(* Logix 5000 project; controller Reto2 vendor 1 type 14 code 156 rev 30.11; software revision 30.00 *)

TASK MainTask (continuous, watchdog 500 ms) : MainProgram

MODULES
   Local : vendor 1 type 14 code 156 (Compact 0, rev 30.11)
      Digital_IN : 1769-IQ16 (Compact 4, rev 1.1, Input RPI 20 ms)
      Digital_OUT : vendor 1 type 7 code 86 (Compact 5, rev 2.1, Output RPI 20 ms)
END_MODULES

VAR_GLOBAL   (* controller tags *)
   AUTO : BOOL;   // Switch Auto FactoryIO
   BOX_AT_ENTRY : BOOL := 1;   // Sensor cajas FactoryIO
   BOX_FEEDER : BOOL;   // Banda 1 cajas FactoryIO
   CLAMP : BOOL;   // Palanca junta cajas FactoryIO
   CLAMPED : BOOL;   // Sensor limite juntador FactoryIO
   Contador1 : COUNTER := (PRE := 2);
   Contador2 : COUNTER := (PRE := 3, ACC := 1);
   Contador3 : COUNTER := (PRE := 3);
   Contador4 : COUNTER := (PRE := 2);
   CONTADOR_CAJAS : DINT;   // Display contador FactoryIO
   CONTADOR_PALLETS : DINT;
   CONTRAER_DE : ALIAS FOR Local:5:O.Data.5;   // Piston Doble efecto Contraer Fisico
   ELEVATOR_DOWN : BOOL;   // Bajar elevador FactoryIO
   ELEVATOR_MOVING : BOOL;   // Sensor movimiento elevador FactoryIO
   ELEVATOR_UP : BOOL;   // Subir elevador FactoryIO
   EMERGENCY_STOP_FACTORY : BOOL := 1;   // Boton stop emergency FactoryIO
   EXIT_CONVEYOR : BOOL;   // Banda 3 Pallet FactoryIO
   EXTENDER_DE : ALIAS FOR Local:5:O.Data.4;   // Piston Doble efecto Extender Fisico
   EXTENDER_SE : ALIAS FOR Local:5:O.Data.6;   // Piston Simple Efecto Fisico
   LOAD_BELT : BOOL;   // Banda 2 cajas FactoryIO
   LOAD_PALLET : BOOL;   // Banda 2 Pallet FactoryIO
   MANUAL : BOOL;   // Switch Manual FactoryIO
   MOTORAC_FISICO : ALIAS FOR Local:5:O.Data.0;   // Motor AC Fisico
   MOVE_TO_LIMIT : BOOL;   // Mover elevador al limite FactoryIO
   OPEN_PLATE : BOOL := 1;   // Trampilla cajas FactoryIO
   osf1 : BOOL;
   osf11 : BOOL;
   osf2 : BOOL;
   osr3 : BOOL;
   PALLET_ENTRY : BOOL := 1;   // Sensor 1 Pallet FactoryIO
   PALLET_EXIT : BOOL := 1;   // Sensor 2 Pallet FactoryIO
   PALLET_FEEDER : BOOL;   // Banda 1 Pallet FactoryIO
   PALLET_LOADED : BOOL;
   PAUSED_FACTORYIO : BOOL;   // Pausando Sim FactoryIO
   PLATE_LIMIT : BOOL := 1;   // Sensor limite compuerta FactoryIO
   PUSH : BOOL;   // Palanca empuja cajas Fisico
   PUSHER_LIMIT : BOOL := 1;   // Sensor limite empujador FactoryIO
   q : BOOL := 1;
   RESET_FACTORYIO : BOOL;   // Boton reset FactoryIO
   RUNNING_FACTORYIO : BOOL := 1;   // Ejecutando Sim FactoryIO
   sb1 : BOOL;
   sb2 : BOOL;
   st3 : BOOL;
   START_FACTORYIO : BOOL;   // Boton verde FactoryIO
   START_FISICO : BOOL;   // Boton verde Fisico
   START_SCADA : BOOL;   // Boton verde SCADA
   STOP_FACTORYIO : BOOL := 1;   // Boton rojo FactoryIO
   STOP_FISICO : BOOL;   // Boton rojo Fisico
   STOP_SCADA : BOOL;   // Boton rojo SCADA
   Temp : BOOL;
   timer1 : TIMER := (PRE := 2500);
   timer2 : TIMER := (PRE := 500);
   TURN : BOOL;   // Palanca girar cajas FactoryIO
   WARNING_LIGHT : BOOL;   // Luces advertencia FactoryIO
   X : BOOL;
   Y : BOOL;
END_VAR

PROGRAM MainProgram   (* main routine MainRoutine *)

ROUTINE Cajas_horizontales   (* ladder *)
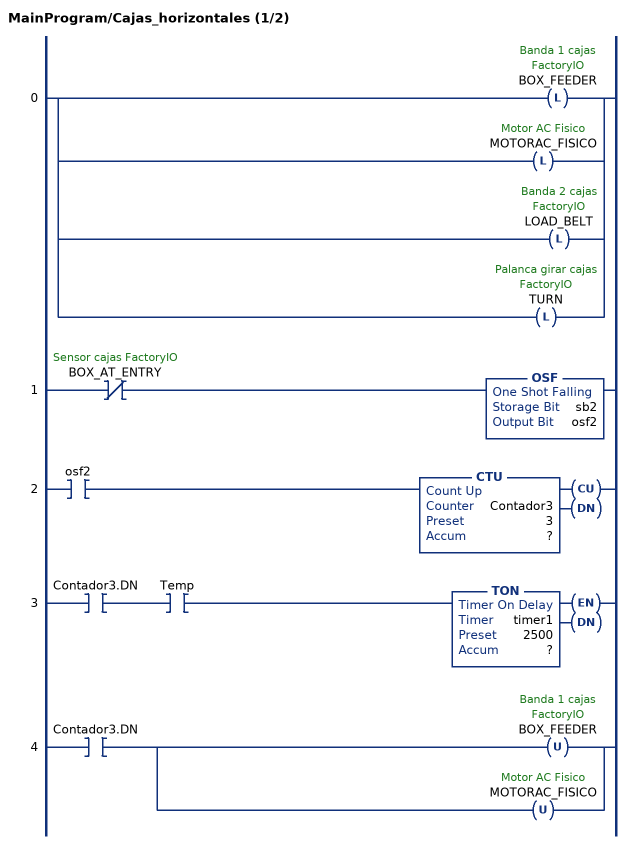
   0: [[[OTL(BOX_FEEDER) ,OTL(MOTORAC_FISICO) ] ,OTL(LOAD_BELT) ] ,OTL(TURN) ];
   1: XIO(BOX_AT_ENTRY)OSF(sb2,osf2);
   2: XIC(osf2)CTU(Contador3,?,?);
   3: XIC(Contador3.DN)XIC(Temp)TON(timer1,?,?);
   4: XIC(Contador3.DN)[OTU(BOX_FEEDER) ,OTU(MOTORAC_FISICO) ];
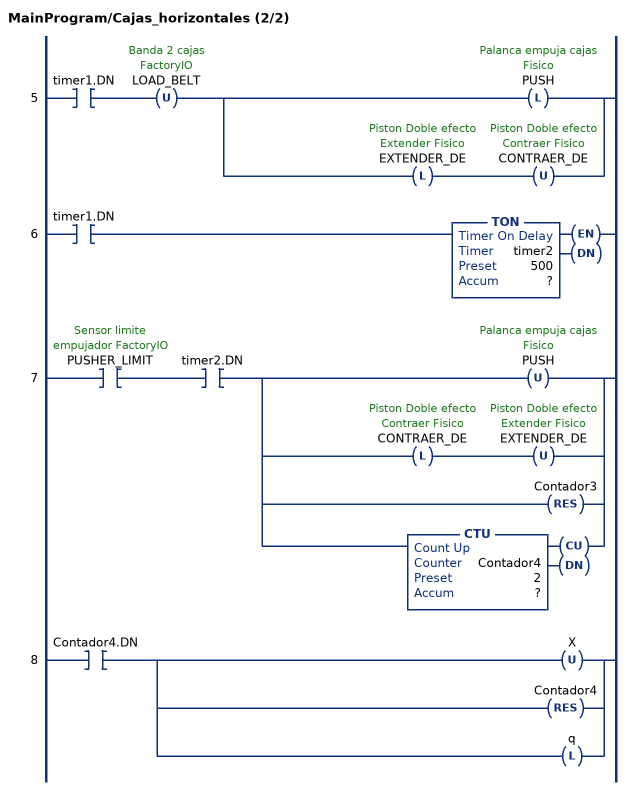
   5: XIC(timer1.DN)OTU(LOAD_BELT)[OTL(PUSH) ,OTL(EXTENDER_DE) OTU(CONTRAER_DE) ];
   6: XIC(timer1.DN)TON(timer2,?,?);
   7: XIC(PUSHER_LIMIT)XIC(timer2.DN)[[[OTU(PUSH) ,OTL(CONTRAER_DE) OTU(EXTENDER_DE) ] ,RES(Contador3) ] ,CTU(Contador4,?,?) ];
   8: XIC(Contador4.DN)[[OTU(X) ,RES(Contador4) ] ,OTL(q) ];
END_ROUTINE

ROUTINE Cajas_verticales   (* ladder *)
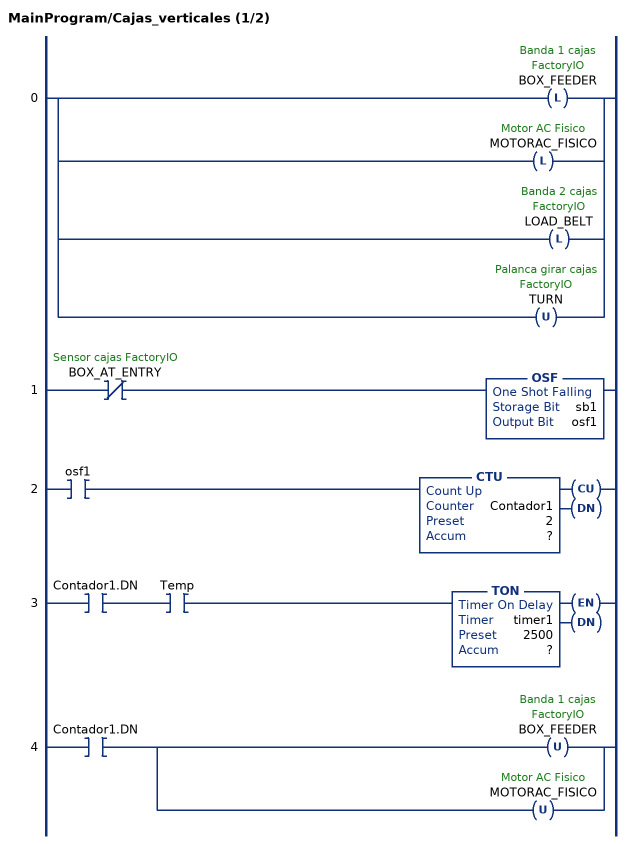
   0: [[[OTL(BOX_FEEDER) ,OTL(MOTORAC_FISICO) ] ,OTL(LOAD_BELT) ] ,OTU(TURN) ];
   1: XIO(BOX_AT_ENTRY)OSF(sb1,osf1);
   2: XIC(osf1)CTU(Contador1,?,?);
   3: XIC(Contador1.DN)XIC(Temp)TON(timer1,?,?);
   4: XIC(Contador1.DN)[OTU(BOX_FEEDER) ,OTU(MOTORAC_FISICO) ];
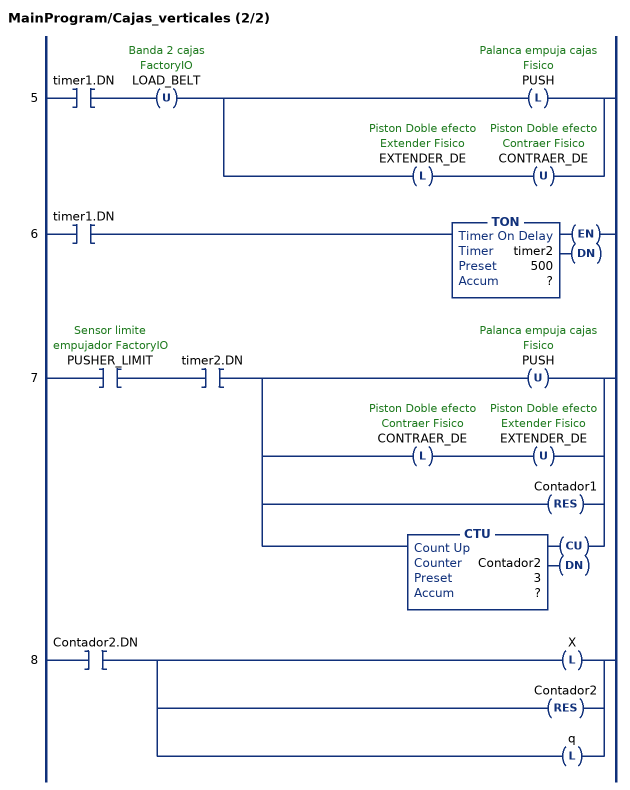
   5: XIC(timer1.DN)OTU(LOAD_BELT)[OTL(PUSH) ,OTL(EXTENDER_DE) OTU(CONTRAER_DE) ];
   6: XIC(timer1.DN)TON(timer2,?,?);
   7: XIC(PUSHER_LIMIT)XIC(timer2.DN)[[[OTU(PUSH) ,OTL(CONTRAER_DE) OTU(EXTENDER_DE) ] ,RES(Contador1) ] ,CTU(Contador2,?,?) ];
   8: XIC(Contador2.DN)[[OTL(X) ,RES(Contador2) ] ,OTL(q) ];
END_ROUTINE

ROUTINE MainRoutine   (* ladder *)
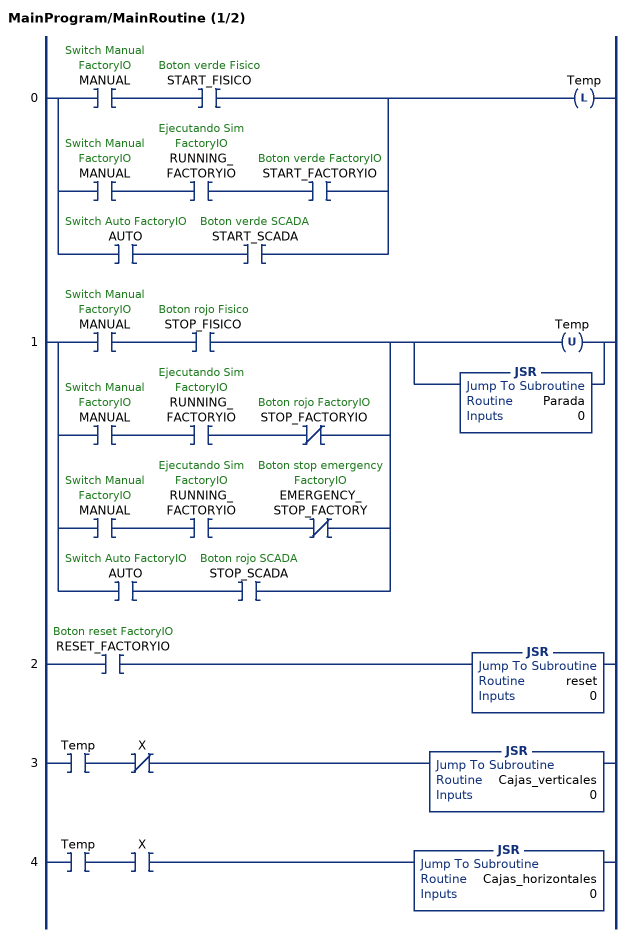
   0: [XIC(MANUAL) XIC(START_FISICO) ,[XIC(MANUAL) XIC(RUNNING_FACTORYIO) XIC(START_FACTORYIO) ,XIC(AUTO) XIC(START_SCADA) ] ]OTL(Temp);
   1: [XIC(MANUAL) XIC(STOP_FISICO) ,[[XIC(MANUAL) XIC(RUNNING_FACTORYIO) XIO(STOP_FACTORYIO) ,XIC(MANUAL) XIC(RUNNING_FACTORYIO) XIO(EMERGENCY_STOP_FACTORY) ] ,XIC(AUTO) XIC(STOP_SCADA) ] ][OTU(Temp) ,JSR(Parada,0) ];
   2: XIC(RESET_FACTORYIO)JSR(reset,0);
   3: XIC(Temp)XIO(X)JSR(Cajas_verticales,0);
   4: XIC(Temp)XIC(X)JSR(Cajas_horizontales,0);
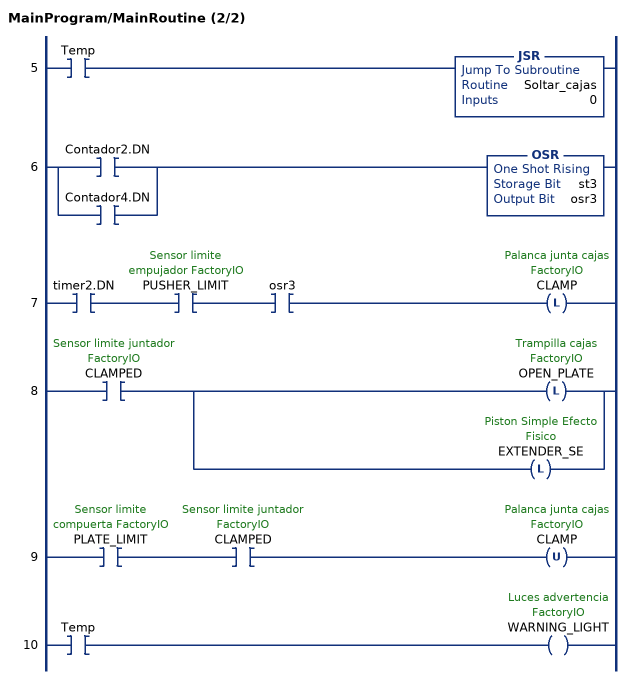
   5: XIC(Temp)JSR(Soltar_cajas,0);
   6: [XIC(Contador2.DN) ,XIC(Contador4.DN) ]OSR(st3,osr3);
   7: XIC(timer2.DN)XIC(PUSHER_LIMIT)XIC(osr3)OTL(CLAMP);
   8: XIC(CLAMPED)[OTL(OPEN_PLATE) ,OTL(EXTENDER_SE) ];
   9: XIC(PLATE_LIMIT)XIC(CLAMPED)OTU(CLAMP);
   10: XIC(Temp)OTE(WARNING_LIGHT);
END_ROUTINE

ROUTINE Parada   (* ladder *)
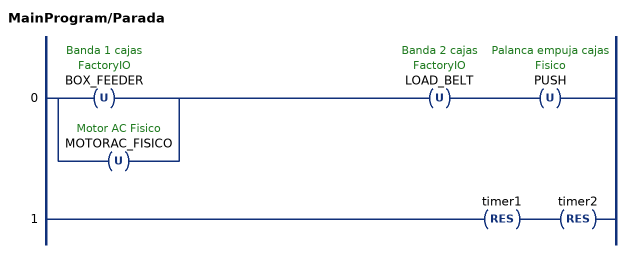
   0: [OTU(BOX_FEEDER) ,OTU(MOTORAC_FISICO) ]OTU(LOAD_BELT)OTU(PUSH);
   1: RES(timer1)RES(timer2);
END_ROUTINE

ROUTINE reset   (* ladder *)
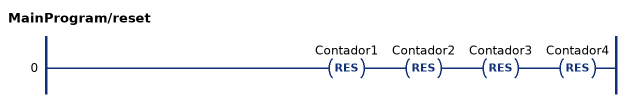
   0: RES(Contador1)RES(Contador2)RES(Contador3)RES(Contador4);
END_ROUTINE

ROUTINE Soltar_cajas   (* ladder *)
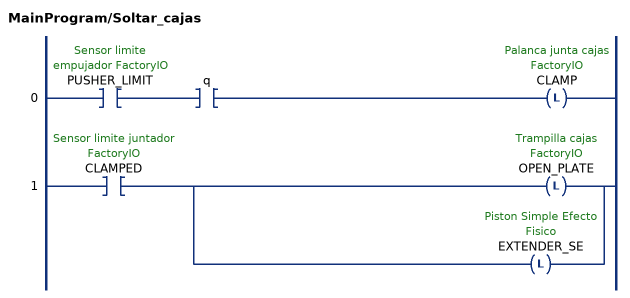
   0: XIC(PUSHER_LIMIT)XIC(q)OTL(CLAMP);
   1: XIC(CLAMPED)[OTL(OPEN_PLATE) ,OTL(EXTENDER_SE) ];
END_ROUTINE
END_PROGRAM
